TYPE ST_Esimerkki :
STRUCT
	
	// Tähän structiin kerätään kaikki Esimerkkitoiminnot, jos niitä on useampia. Helpottaa HMI toimintoja.
	
	stEsimerkki_1			: ST_EsimerkkiHMI;
	stEsimerkki_2			: ST_EsimerkkiHMI;
END_STRUCT
END_TYPE

(* stored: Version 1.1.0.1
   DUT ST_Esimerkki: Id {4b75c15f-4245-4007-bca7-965f4c534882} *)
